// TIA Portal V20 export
TYPE "Fault"
// stored: Access Published, Namespace Global
   STRUCT
      Motor_Error : Bool;
      Sensor_Blockage : Bool;
   END_STRUCT;
END_TYPE
